// TIA Portal V17 export
// export: Created 2024-08-09T12:53:24.7337085Z, ExportSetting WithDefaults, DisplayName Totally Integrated Automation Portal, DisplayVersion V17 Update 7, DisplayName TIA Portal Openness, DisplayVersion V17 Update 7, DisplayName TIA Portal Version Control Interface, DisplayVersion V17, DisplayName STEP 7 Professional, DisplayVersion V17 Update 7, DisplayName STEP 7 Safety, DisplayVersion V17 Update 6, DisplayName WinCC Professional, DisplayVersion V17 Update 7
TYPE "S_MODULE_SUIVI_COMMUNENSACH"
// stored: IsFailsafeCompliant false
   STRUCT
      Tab_Lots { ExternalAccessible := 'False'; ExternalVisible := 'False'; ExternalWritable := 'False'} : Array[0.."MAX_LOTS"] of "S_SUIVI_ENSACHAGE";   // Table des zones de suivi lot
   END_STRUCT;
END_TYPE
